(* CoDeSys 2.3.9.37 project: Cap6_7.pro *)
(* Libraries: Standard.lib 4.10.05 12:14:46 *)

(* Global variable list: Global_Variables *)
VAR_GLOBAL

      (* Entradas *)
      START:BOOL;
	A:BOOL;
	B:BOOL;
      (* Salidas *)
	MOTOR_IZ:BOOL;
	MOTOR_DE:BOOL;

      (* Variable para la simulación
         de la animación *)
	Vel:INT:=1;
END_VAR

(* POU PLC_PRG, FBD *)
PROGRAM PLC_PRG
VAR

END_VAR
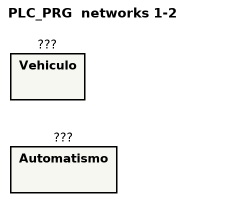
_FBD_ (* Function Block Diagram *)
NETWORK 1
	???:Vehiculo()
NETWORK 2
	???:Automatismo()
_END_FBD_
END_PROGRAM

(* POU Vehiculo, ST *)
PROGRAM Vehiculo
VAR
	PosX: INT;
END_VAR
A:=FALSE;
B:=FALSE;


IF MOTOR_DE=TRUE THEN

     PosX:=PosX+Vel;

END_IF

IF MOTOR_IZ=TRUE THEN

     PosX:=PosX-Vel;

END_IF


IF PosX<=0 THEN
   A:=TRUE;
END_IF

IF PosX>=400 THEN
  B:=TRUE;
END_IF
END_PROGRAM

(* POU Automatismo, LD *)
PROGRAM Automatismo
VAR
	Re: BOOL;
	Der: BOOL;
	Izq: BOOL;
END_VAR
VAR (* helpers for the ST form of the networks *)
	_p1 : BOOL;
	_p2 : BOOL;
	_p3 : BOOL;
END_VAR
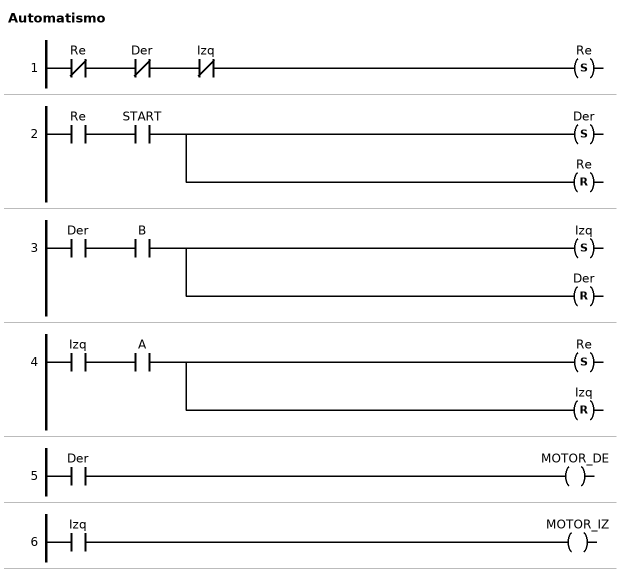
_LD_ (* Ladder Diagram *)
NETWORK 1
	[/Re] - [/Der] - [/Izq] --- (S Re)
NETWORK 2
	[Re] - [START] --- (S Der) (R Re)
NETWORK 3
	[Der] - [B] --- (S Izq) (R Der)
NETWORK 4
	[Izq] - [A] --- (S Re) (R Izq)
NETWORK 5
	[Der] --- (MOTOR_DE)
NETWORK 6
	[Izq] --- (MOTOR_IZ)
_END_LD_
(* the same logic as Structured Text *)
(* Network 1 *)
IF NOT Re AND NOT Der AND NOT Izq THEN Re := TRUE; END_IF;
(* Network 2 *)
_p1 := Re AND START;
IF _p1 THEN Der := TRUE; Re := FALSE; END_IF;
(* Network 3 *)
_p2 := Der AND B;
IF _p2 THEN Izq := TRUE; Der := FALSE; END_IF;
(* Network 4 *)
_p3 := Izq AND A;
IF _p3 THEN Re := TRUE; Izq := FALSE; END_IF;
(* Network 5 *)
MOTOR_DE := Der;
(* Network 6 *)
MOTOR_IZ := Izq;
END_PROGRAM

(* Visualisation Vehiculo
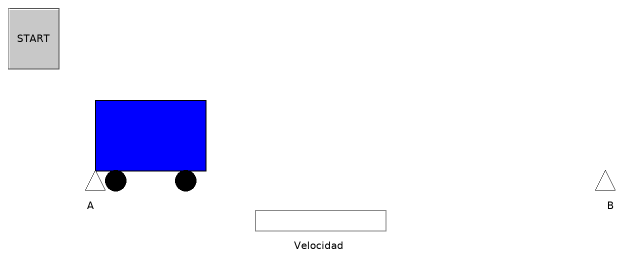
rectangle at (140,120)-(251,191): x offset Vehiculo.PosX
polygon at (130,190)-(150,210): alarm colour if .A
polygon at (640,190)-(660,210): alarm colour if .B
button at (53,28)-(104,89): text "START"; toggles START
ellipse at (150,190)-(171,211): x offset Vehiculo.PosX
ellipse at (220,190)-(241,211): x offset Vehiculo.PosX
rectangle at (310,250)-(421,281): text "Velocidad"
rectangle at (80,210)-(191,241): text "A"
rectangle at (600,210)-(711,241): text "B"
1 more shapes without text or variables
*)
